//{attribute 'qualified_only'}
//{attribute 'strict'}
{attribute 'to_string'}
TYPE E_ElevatorState :
(
	//Idle,
    MovingUp,
    MovingDown,
    DoorControl
	//Fault
);
END_TYPE

(* stored: Version 1.1.0.1
   DUT E_ElevatorState: Id {eb632649-71c8-4fbc-ab50-572192c7ac77} *)
